// SIMATIC STEP 7 (V5.x) project TEMA 13 EJERCICIO 38
// CPU: CPU313 C-2 DP(1)
// station: P_ADR_BUS
// station: Hardware
// station: Equipo SIMATIC 300
// program: Programa S7(1)

SYMBOL_TABLE
""		
"FLANCOS"	DB 1	DB 1
"P MARCHA"	I 0.0	BOOL
"FC 2 ABAJO"	I 0.1	BOOL
"FC 3 ARRIBA"	I 0.2	BOOL
"FC 4 IZQUIERDA"	I 0.3	BOOL
"FC 5 DERECHA"	I 0.4	BOOL
"CONTROL"	MB 1	BYTE
"Cycle Execution"	OB 1	OB 1
"SUBIR"	Q 0.0	BOOL
"BAJAR"	Q 0.1	BOOL
"DERECHA"	Q 0.2	BOOL
"IZQUIERDA"	Q 0.3	BOOL
END_SYMBOL_TABLE

DATA_BLOCK "FLANCOS"	// DB 1
VERSION : 0.1
  STRUCT
   M0 : BOOL ;
   M1 : BOOL ;
   M2 : BOOL ;
   M3 : BOOL ;
   M4 : BOOL ;
   M5 : BOOL ;
   M6 : BOOL ;
   M7 : BOOL ;
   M10 : BOOL ;
   M11 : BOOL ;
   M12 : BOOL ;
   M13 : BOOL ;
   M14 : BOOL ;
   M15 : BOOL ;
   M16 : BOOL ;
   M17 : BOOL ;
  END_STRUCT ;	
BEGIN
END_DATA_BLOCK

ORGANIZATION_BLOCK "Cycle Execution"	// OB 1
TITLE = "Main Program Sweep (Cycle)"
//PROCESO CICLICO CON CRUA.
VERSION : 0.1
VAR_TEMP
  OB1_EV_CLASS : BYTE ;	//Bits 0-3 = 1 (Coming event), Bits 4-7 = 1 (Event class 1)
  OB1_SCAN_1 : BYTE ;	//1 (Cold restart scan 1 of OB 1), 3 (Scan 2-n of OB 1)
  OB1_PRIORITY : BYTE ;	//Priority of OB Execution
  OB1_OB_NUMBR : BYTE ;	//1 (Organization block 1, OB1)
  OB1_RESERVED_1 : BYTE ;	//Reserved for system
  OB1_RESERVED_2 : BYTE ;	//Reserved for system
  OB1_PREV_CYCLE : INT ;	//Cycle time of previous OB1 scan (milliseconds)
  OB1_MIN_CYCLE : INT ;	//Minimum cycle time of OB1 (milliseconds)
  OB1_MAX_CYCLE : INT ;	//Maximum cycle time of OB1 (milliseconds)
  OB1_DATE_TIME : DATE_AND_TIME ;	//Date and time OB1 started
END_VAR
BEGIN
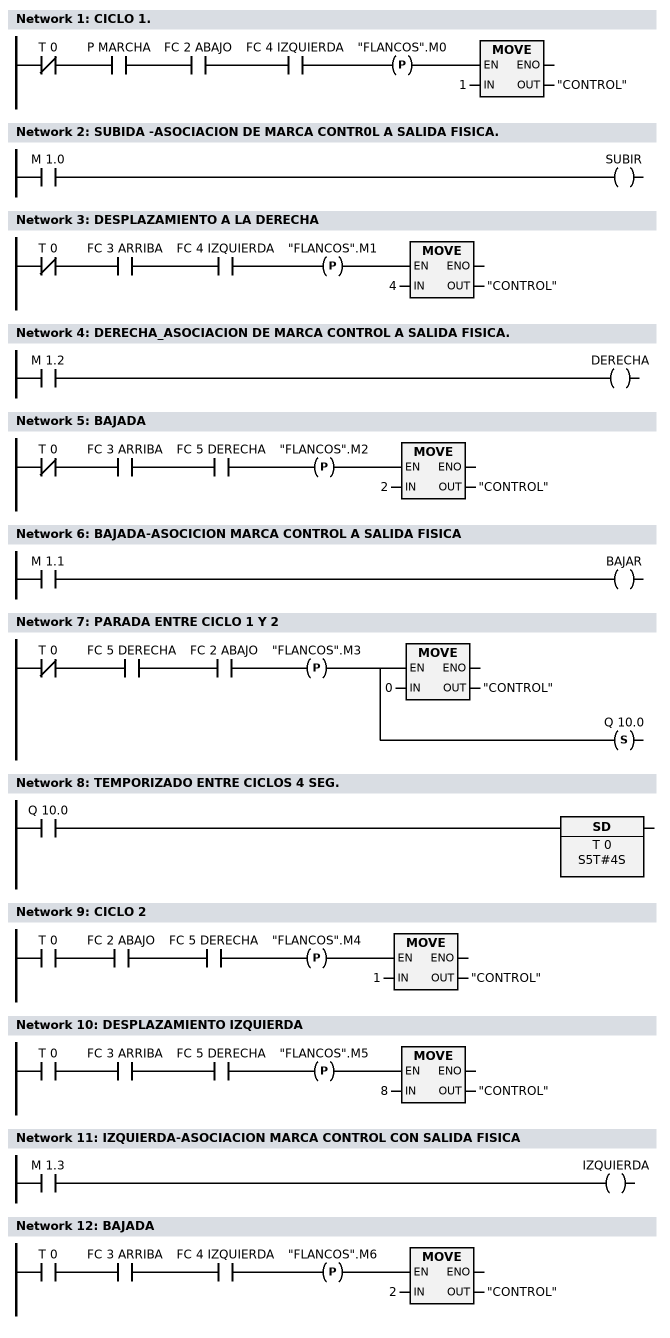
NETWORK
TITLE = CICLO 1.
//PUESTA EN MARCHA-SUBIDA DE GANCHO
      AN    T 0;
      A     "P MARCHA";
      A     "FC 2 ABAJO";
      A     "FC 4 IZQUIERDA";
      FP    "FLANCOS".M0;
      JNB   _001;
      L     1;
      T     "CONTROL";
_001: NOP   0;
NETWORK
TITLE = SUBIDA -ASOCIACION DE MARCA CONTR0L A SALIDA FISICA.
      A     M 1.0;
      =     "SUBIR";
NETWORK
TITLE = DESPLAZAMIENTO A LA DERECHA
      AN    T 0;
      A     "FC 3 ARRIBA";
      A     "FC 4 IZQUIERDA";
      FP    "FLANCOS".M1;
      JNB   _002;
      L     4;
      T     "CONTROL";
_002: NOP   0;
NETWORK
TITLE = DERECHA_ASOCIACION DE MARCA CONTROL A SALIDA FISICA.
      A     M 1.2;
      =     "DERECHA";
NETWORK
TITLE = BAJADA
      AN    T 0;
      A     "FC 3 ARRIBA";
      A     "FC 5 DERECHA";
      FP    "FLANCOS".M2;
      JNB   _003;
      L     2;
      T     "CONTROL";
_003: NOP   0;
NETWORK
TITLE = BAJADA-ASOCICION MARCA CONTROL A SALIDA FISICA
      A     M 1.1;
      =     "BAJAR";
NETWORK
TITLE = PARADA ENTRE CICLO 1 Y 2 
      AN    T 0;
      A     "FC 5 DERECHA";
      A     "FC 2 ABAJO";
      FP    "FLANCOS".M3;
      =     L 20.0;
      A     L 20.0;
      JNB   _004;
      L     0;
      T     "CONTROL";
_004: NOP   0;
      A     L 20.0;
      BLD   102;
      S     Q 10.0;
NETWORK
TITLE = TEMPORIZADO ENTRE CICLOS 4 SEG.
//EN EL PRIMER CICLO COLOCO UN CERRADO DE TO EN CADA LINEA DE ACCIONMIENTO POR 
//SEGURIDAD EVITANDO QUE EN UN CASO REMOTO ACCTIVE OTRA MOV-E.
//EN EL SEGUNDO CICLO EL CONTACTO SERA ABIERTO PARA GOBERNAR Y DIFERENCIAR EN 
//CASOS QUE COINCIDAN LAS PAUTAS DE ACCIONMIENTO.
      A     Q 10.0;
      L     S5T#4S;
      SD    T 0;
NETWORK
TITLE = CICLO 2 
//SUBIDA TEMPORIZADA
      A     T 0;
      A     "FC 2 ABAJO";
      A     "FC 5 DERECHA";
      FP    "FLANCOS".M4;
      JNB   _005;
      L     1;
      T     "CONTROL";
_005: NOP   0;
NETWORK
TITLE = DESPLAZAMIENTO IZQUIERDA
      A     T 0;
      A     "FC 3 ARRIBA";
      A     "FC 5 DERECHA";
      FP    "FLANCOS".M5;
      JNB   _006;
      L     8;
      T     "CONTROL";
_006: NOP   0;
NETWORK
TITLE = IZQUIERDA-ASOCIACION MARCA CONTROL CON SALIDA FISICA
      A     M 1.3;
      =     "IZQUIERDA";
NETWORK
TITLE = BAJADA 
      A     T 0;
      A     "FC 3 ARRIBA";
      A     "FC 4 IZQUIERDA";
      FP    "FLANCOS".M6;
      JNB   _007;
      L     2;
      T     "CONTROL";
_007: NOP   0;
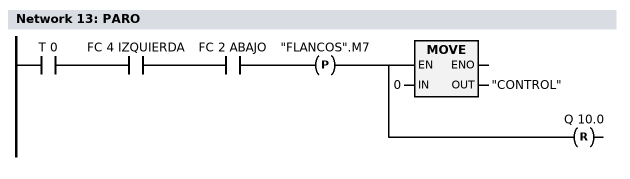
NETWORK
TITLE = PARO 
      A     T 0;
      A     "FC 4 IZQUIERDA";
      A     "FC 2 ABAJO";
      FP    "FLANCOS".M7;
      =     L 20.0;
      A     L 20.0;
      JNB   _008;
      L     0;
      T     "CONTROL";
_008: NOP   0;
      A     L 20.0;
      BLD   102;
      R     Q 10.0;
END_ORGANIZATION_BLOCK
